// TIA Portal V17 export
// export: Created 2024-08-09T12:53:23.9389727Z, ExportSetting WithDefaults, DisplayName Totally Integrated Automation Portal, DisplayVersion V17 Update 7, DisplayName TIA Portal Openness, DisplayVersion V17 Update 7, DisplayName TIA Portal Version Control Interface, DisplayVersion V17, DisplayName STEP 7 Professional, DisplayVersion V17 Update 7, DisplayName STEP 7 Safety, DisplayVersion V17 Update 6, DisplayName WinCC Professional, DisplayVersion V17 Update 7
TYPE "S_SuiviCommunCharg"
// stored: IsFailsafeCompliant false
   STRUCT
      _TabLots { S7_SetPoint := 'True'} : Array[0.."MAX_LOTS"] of "S_SuiviCommande";
      _NoLot { ExternalAccessible := 'False'; ExternalVisible := 'False'; ExternalWritable := 'False'} : USInt;   // no de lot pour gestion couleurs
   END_STRUCT;
END_TYPE
